// TIA Portal V16 export
// export: Created 2024-03-27T10:04:38.1489128Z, ExportSetting WithDefaults, DisplayName Totally Integrated Automation Portal, DisplayVersion V16, DisplayName TIA Portal Version Control Interface, DisplayVersion V16, DisplayName TIA Portal Openness, DisplayVersion V16, DisplayName STEP 7 Professional, DisplayVersion V16, DisplayName STEP 7 Safety, DisplayVersion V16, DisplayName WinCC Advanced, DisplayVersion V16
TYPE "UR__T2O_IOs"
// stored: IsFailsafeCompliant false
   STRUCT
      "Standard digital inputs" : USInt;
      "Configurable digital inputs" : USInt;
      "Standard digital outputs" : USInt;
      "Configurable digital outputs" : USInt;
      "Analog I/O types" : USInt;
      Reserved_8_15 { ExternalAccessible := 'False'; ExternalVisible := 'False'; ExternalWritable := 'False'} : USInt;
      Reserved_16_31 { ExternalAccessible := 'False'; ExternalVisible := 'False'; ExternalWritable := 'False'} : UInt;
      "Standard analog input [A or V]" : Array[0..1] of Real;
      "Standard analog output [A or V]" : Array[0..1] of Real;
      "I/O current [A]" : Real;
      "Euromap67 input bits" : Array[0..31] of Bool;
      "Euromap67 output bits" : Array[0..31] of Bool;
      "Euromap67 24V voltage" : Real;
      "Euromap67 24V current" : Real;
   END_STRUCT;
END_TYPE
